(* IEC 61131-3 sources: CodesysTest/export/Function Blocks/SolenoidValves/FB_PneumaticActuator.pou/ExtendAsserted.prop, 1 file *)

(* ---- Get.pm.st ---- *)
(*#-#-#-#-#-#-#-#-#-#---Declaration---#-#-#-#-#-#-#-#-#-#-#-#-#*)

VAR
END_VAR
(*#-#-#-#-#-#-#-#-#-#---Implementation---#-#-#-#-#-#-#-#-#-#-#-#-#*)

ExtendAsserted := _extendAsserted;
